FUNCTION_BLOCK RunMaterial
VAR_INPUT
END_VAR
VAR_OUTPUT
END_VAR
VAR
	header AT%M* : MaterialHeader;
	block AT%M* : MaterialBlock;
END_VAR
VAR PERSISTENT
	isNotLinked : bool; //if not linked , do not handshaking
END_VAR

PROPERTY Act : bool
GET
Act := header.wordOut.1;
END_GET
SET
IF isNotLinked THEN
	return;
END_IF

header.wordOut.1 := Act;
END_SET
END_PROPERTY

PROPERTY Data : MaterialBlock
GET
Data := block;
END_GET
SET
block := Data;
END_SET
END_PROPERTY

PROPERTY Id : DWORD
GET
Id := header.id;
END_GET
SET
header.id := Id;
END_SET
END_PROPERTY

PROPERTY Valid : bool
GET
Valid := header.wordOut.2;
END_GET
SET
header.wordOut.2 := Valid;
END_SET
END_PROPERTY

END_FUNCTION_BLOCK

(* stored: Version 1.1.0.1, ProductVersion 3.1.4022.10
   POU RunMaterial: Id {9073517c-3b61-4b10-a156-8338bfb2c574}, SpecialFunc None
   Property Act: Id {236bb699-4edc-4d48-a62f-bc4ddb0aabdf}
   Get Get: Id {579db0b6-a439-4489-af03-b8d193df4417}
   Set Set: Id {d98760fd-3777-4f25-8402-51e31ca98d9b}
   Property Data: Id {79a915a5-cf76-4b51-8c57-c4d23e98aa43}
   Get Get: Id {83a4552a-77c4-4f9d-9bfa-8112928f18d9}
   Set Set: Id {0928f0d4-1ea0-4c84-980c-5f4b4a3fc0c4}
   Property Id: Id {76cc9878-8344-4469-85c7-4021594103e7}
   Get Get: Id {52057c29-0d31-4150-8be7-d3db7c8824a2}
   Set Set: Id {4db29320-7c5f-4cee-bfd1-83007f696f64}
   Property Valid: Id {81a23da7-5efb-49a3-9451-5b7d459a1adb}
   Get Get: Id {d2210c58-6905-4049-a4ca-7630c9005422}
   Set Set: Id {4d838795-a156-4765-b1a6-c8dafa3a1944} *)
